TYPE ST_FireDetection_get_1 :
STRUCT
	SmokeDetectors : ST_SmokeDetectors;
	CODetectors	:	ST_CODetectors;
	
	Events	:	ST_FireSystem_Events;
END_STRUCT
END_TYPE

(* stored: Version 1.1.0.1, ProductVersion 3.1.4024.12
   DUT ST_FireDetection_get_1: Id {54ea5c58-00fb-436d-b0eb-260a3a71f4b7} *)
